FUNCTION_BLOCK Test_TStringSplitter_Splits_On_Tab EXTENDS T_UnitTestBase
VAR
    StringSplitter : T_StringSplitter;
END_VAR

METHOD Init
VAR_INPUT
END_VAR
END_METHOD

{attribute 'analysis' := '-33'} // inhibit unused variable warning
METHOD RunTest

StringSplitter.Init(Str    := 'Bob$TCharles$TDavid',
                    Delim1 := '$T',
                    Delim2 := '');

AssertEquals_STRING(Expected := 'Bob',
                    Actual   := StringSplitter.GetNext(),
                    Message  := 'StringSplitter.GetNext()');

AssertEquals_STRING(Expected := 'Charles',
                    Actual   := StringSplitter.GetNext(),
                    Message  := 'StringSplitter.GetNext()');

AssertEquals_STRING(Expected := 'David',
                    Actual   := StringSplitter.GetNext(),
                    Message  := 'StringSplitter.GetNext()');

TestCompleted := TRUE;
END_METHOD

END_FUNCTION_BLOCK

(* stored: Version 1.1.0.1, ProductVersion 3.1.4024.12
   POU Test_TStringSplitter_Splits_On_Tab: Id {86e3e891-db36-057f-3764-d41869894fb8}, SpecialFunc None
   Method Init: Id {490dfb9f-1b3e-099b-3ad2-ef0779468e82}
   Method RunTest: Id {02fbd306-982e-0b16-2e18-81ef9210825c} *)
